FUNCTION_BLOCK fb_Blink
VAR_INPUT
END_VAR
VAR_OUTPUT
END_VAR
VAR
		t1 : TON;
		t2 : TON;
END_VAR




t1.IN := (t2.Q = FALSE);

t2.IN := t1.Q;


t1(PT:=t#1s);
t2(PT:=t#2s);

END_FUNCTION_BLOCK

(* stored: Version 1.1.0.1, ProductVersion 3.1.4024.0
   POU fb_Blink: Id {4b382ce4-3218-4416-9ced-7864c2b52936}, SpecialFunc None *)
